Omron CX-Programmer project NewProject (CX-Programmer 9.03)

# PLC CLP: CJ1M CPU11
I/O table (CPU CJ1M-CPU11): rack 0 slot 0 CJ1W-ETN21(ETN11Mode); rack 0 slot 1 CJ1W-ID211; rack 0 slot 2 CJ1W-OD211; rack 0 slot 3 CJ1W-ID211; rack 0 slot 4 CJ1W-OD211; rack 0 slot 5 CJ1W-ID211; rack 0 slot 6 CJ1W-OD232

## Global symbols (name address type ; comment)
AS_RS_Ativado 5.02 BOOL
AS_RS_Eixo_X_Ctrg 5.04 BOOL
AS_RS_Eixo_X_D0 5.05 BOOL
AS_RS_Eixo_X_D1 5.06 BOOL
AS_RS_Eixo_X_D2 5.07 BOOL
AS_RS_Eixo_X_D3 5.08 BOOL
AS_RS_Eixo_X_To_Home 5.03 BOOL
AS_RS_Eixo_Y_Ctrg 5.10 BOOL
AS_RS_Eixo_Y_D0 5.11 BOOL
AS_RS_Eixo_Y_D1 5.12 BOOL
AS_RS_Eixo_Y_D2 5.13 BOOL
AS_RS_Eixo_Y_D3 5.14 BOOL
AS_RS_Eixo_Y_To_Home 5.09 BOOL
AS_RS_Eixo_Z_Ctrg 6.00 BOOL
AS_RS_Eixo_Z_D0 6.01 BOOL
AS_RS_Eixo_Z_D1 6.02 BOOL
AS_RS_Eixo_Z_D2 6.03 BOOL
AS_RS_Eixo_Z_D3 6.04 BOOL
AS_RS_Eixo_Z_To_Home 5.15 BOOL
AS_RS_Home_X_Completo 4.05 BOOL
AS_RS_Home_Y_Completo 4.07 BOOL
AS_RS_Home_Z_Completo 4.09 BOOL
AS_RS_Pos_X_Completa 4.04 BOOL
AS_RS_Pos_Y_Completa 4.06 BOOL
AS_RS_Pos_Z_Completa 4.08 BOOL
AUX_CTRG W10.02 BOOL
AUX_X_OK W10.05 BOOL
AUX_X_OK_DESCIDA W16.00 BOOL
AUX_Y_OK W10.07 BOOL
AUX_Z_OK W10.06 BOOL
AUX_Z_OK_DESCIDA W16.01 BOOL
T0005 BOOL  ; 3
CONF_Z W11.05 BOOL
Confirmacao W4.00 BOOL
Eletroval1 1.06 BOOL
Eletroval2 1.07 BOOL
Eletroval3 1.08 BOOL
Eletroval4 1.09 BOOL
Elevar_Z W15.00 BOOL
Esteira1 1.00 BOOL
Esteira2 1.01 BOOL
Esteira3 1.02 BOOL
Esteira4 1.03 BOOL
Etapa BOOL
Etapa0 W0.00 BOOL
Etapa1 W0.01 BOOL
Etapa10 W1.02 BOOL
Etapa11 W1.03 BOOL
Etapa2 W0.02 BOOL
Etapa3 W0.03 BOOL
Etapa4 W0.04 BOOL
Etapa5 W0.05 BOOL
Etapa6 W0.06 BOOL
Etapa7 W0.07 BOOL
Etapa8 W1.00 BOOL
Etapa9 W1.01 BOOL
Home_X_Completo 4.05 BOOL
Home_Y_Completo 4.07 BOOL
Home_Z_Completo 4.09 BOOL
Pos_X_Completa 4.04 BOOL
Pos_Y_Completa 4.06 BOOL
Pos_Z_Completa 4.08 BOOL
Sensor1 0.00 BOOL
Sensor2 0.01 BOOL
Sensor3 0.02 BOOL
Sensor4 0.03 BOOL
X_CTRG 5.04 BOOL
X_D0 5.05 BOOL
X_D1 5.06 BOOL
X_D2 5.07 BOOL
X_D3 5.08 BOOL
X_To_Home 5.03 BOOL
Y_CTRG 5.10 BOOL
Y_D0 5.11 BOOL
Y_D1 5.12 BOOL
Y_D2 5.13 BOOL
Y_D3 5.14 BOOL
Y_To_Home 5.09 BOOL
Z_CTRG 6.00 BOOL
Z_D0 6.01 BOOL
Z_D1 6.02 BOOL
Z_D2 6.03 BOOL
Z_D3 6.04 BOOL
Z_To_Home 5.15 BOOL

## Program NewProgram1 (cyclic task 0)
Local symbols
AS_RS_Ativado 5.02 BOOL
AUX_CTRG W10.02 BOOL
AUX_ESTEIRA_OK W65.00 BOOL
AUX_ROBO_OK W50.00 BOOL
AUX_VISAO_OK W50.01 BOOL
AUX_X_OK W10.05 BOOL
AUX_Y_OK W10.07 BOOL
AUX_Z_OK W10.06 BOOL
Confirmacao W4.00 BOOL
E0_ESTEIRA W60.00 BOOL
E1_ESTEIRA W60.01 BOOL
E2_ESTEIRA W60.02 BOOL
E3_ESTEIRA W60.03 BOOL
E4_ESTEIRA W60.04 BOOL
E5_ESTEIRA W60.05 BOOL
E6_ESTEIRA W60.06 BOOL
E7_ESTEIRA W60.07 BOOL
Eletroval1 1.06 BOOL
Eletroval2 1.07 BOOL
Eletroval3 1.08 BOOL
Eletroval4 1.09 BOOL
Elevar_Z W15.00 BOOL
Esteira1 1.00 BOOL
Esteira2 1.01 BOOL
Esteira3 1.02 BOOL
Esteira4 1.03 BOOL
Etapa BOOL
Etapa0 W0.00 BOOL
Etapa1 W0.01 BOOL
Etapa10 W1.02 BOOL
Etapa11 W1.03 BOOL
Etapa12 W1.04 BOOL
Etapa13 W1.05 BOOL
Etapa14 W1.06 BOOL
Etapa15 W1.07 BOOL
Etapa16 W2.00 BOOL
Etapa17 W2.01 BOOL
Etapa18 W2.02 BOOL
Etapa19 W2.03 BOOL
Etapa2 W0.02 BOOL
Etapa20 W2.04 BOOL
Etapa21 W2.05 BOOL
Etapa22 W2.06 BOOL
Etapa23 W2.07 BOOL
Etapa24 W3.01 BOOL
Etapa25 W3.02 BOOL
Etapa26 W3.03 BOOL
Etapa27 W3.04 BOOL
Etapa28 W3.05 BOOL
Etapa29 W3.06 BOOL
Etapa3 W0.03 BOOL
Etapa30 W3.07 BOOL
Etapa31 W4.01 BOOL
Etapa32 W4.02 BOOL
Etapa33 W4.03 BOOL
Etapa34 W4.04 BOOL
Etapa35 W4.05 BOOL
Etapa36 W4.06 BOOL
Etapa4 W0.04 BOOL
Etapa5 W0.05 BOOL
Etapa6 W0.06 BOOL
Etapa7 W0.07 BOOL
Etapa8 W1.00 BOOL
Etapa9 W1.01 BOOL
FLAG_ROBO W50.02 BOOL
Home_X_Completo 4.05 BOOL
Home_Y_Completo 4.07 BOOL
Home_Z_Completo 4.09 BOOL
INICIA_ESTEIRA BOOL
INICIA_ESTEIRAS W50.05 BOOL
MAO_PEGAR_ARMAZEM 6.08 BOOL
MAO_PEGAR_ESTEIRA 6.09 BOOL
PEGAR_MAO_ESTEIRA BOOL
Pos_X_Completa 4.04 BOOL
Pos_Y_Completa 4.06 BOOL
Pos_Z_Completa 4.08 BOOL
Sensor1 0.00 BOOL
Sensor2 0.01 BOOL
Sensor3 0.02 BOOL
Sensor4 0.03 BOOL
WORD_X W35 WORD
WORD_Z W40 WORD
XD0 BOOL
X_CTRG 5.04 BOOL
X_D0 5.05 BOOL
X_D1 5.06 BOOL
X_D2 5.07 BOOL
X_D3 5.08 BOOL
X_To_Home 5.03 BOOL
Y_CTRG 5.10 BOOL
Y_D0 5.11 BOOL
Y_D1 5.12 BOOL
Y_D2 5.13 BOOL
Y_D3 5.14 BOOL
Y_To_Home 5.09 BOOL
Z_CTRG 6.00 BOOL
Z_D0 6.01 BOOL
Z_D1 6.02 BOOL
Z_D2 6.03 BOOL
Z_D3 6.04 BOOL
Z_To_Home 5.15 BOOL

### Section Armazem

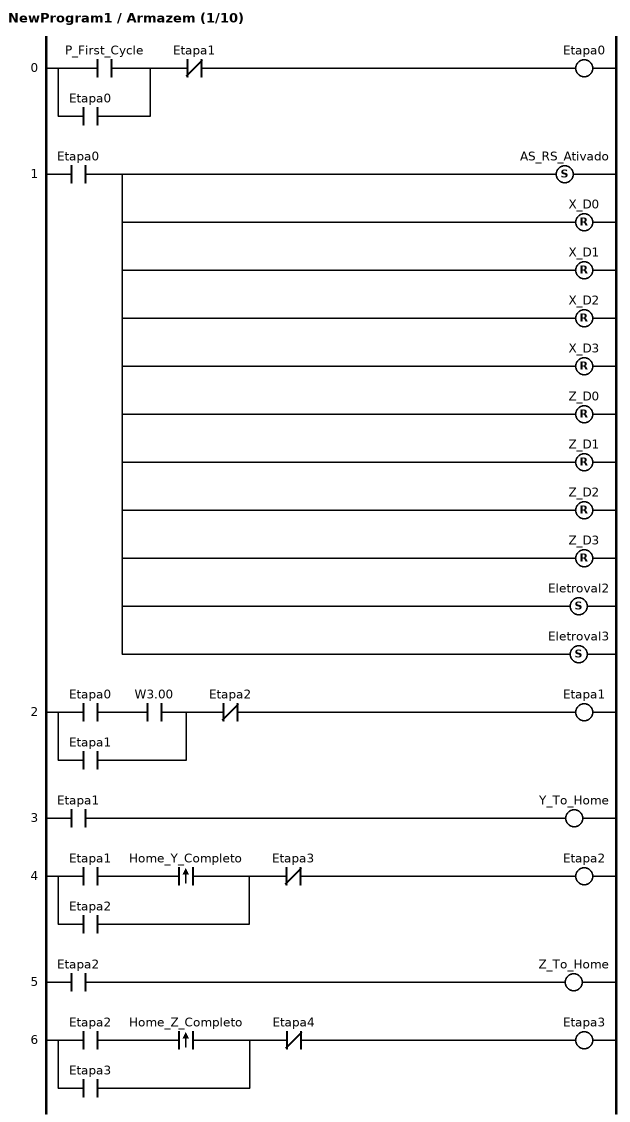
; rung 0
LD P_First_Cycle
OR Etapa0
ANDNOT Etapa1
OUT Etapa0
; rung 1
LD Etapa0
SET AS_RS_Ativado
RSET X_D0
RSET X_D1
RSET X_D2
RSET X_D3
RSET Z_D0
RSET Z_D1
RSET Z_D2
RSET Z_D3
SET Eletroval2
SET Eletroval3
; rung 2
LD Etapa0
AND W3.00
OR Etapa1
ANDNOT Etapa2
OUT Etapa1
; rung 3
LD Etapa1
OUT Y_To_Home
; rung 4
LD Etapa1
@AND Home_Y_Completo
OR Etapa2
ANDNOT Etapa3
OUT Etapa2
; rung 5
LD Etapa2
OUT Z_To_Home
; rung 6
LD Etapa2
@AND Home_Z_Completo
OR Etapa3
ANDNOT Etapa4
OUT Etapa3

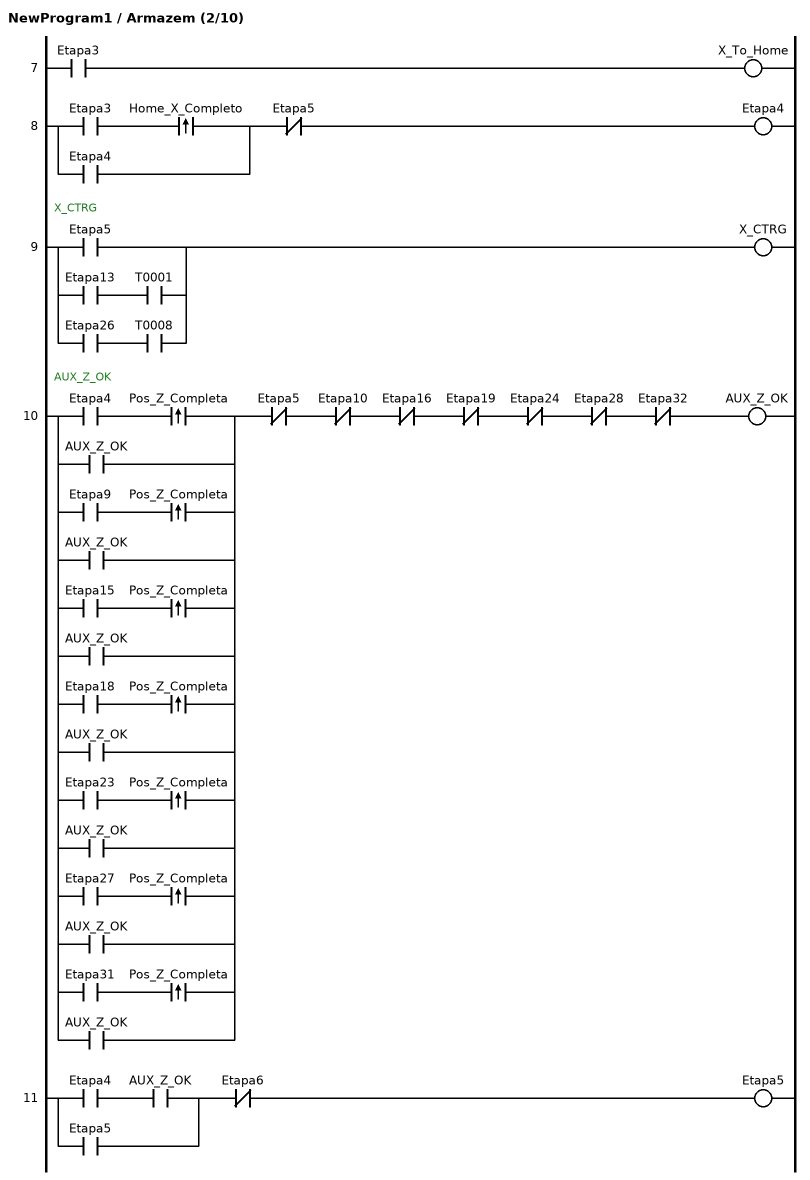
; rung 7
LD Etapa3
OUT X_To_Home
; rung 8
LD Etapa3
@AND Home_X_Completo
OR Etapa4
ANDNOT Etapa5
OUT Etapa4
; rung 9: X_CTRG
LD Etapa5
LD Etapa13
AND T0001
ORLD
LD Etapa26
AND T0008
ORLD
OUT X_CTRG
; rung 10: AUX_Z_OK
LD Etapa4
@AND Pos_Z_Completa
OR AUX_Z_OK
LD Etapa9
@AND Pos_Z_Completa
ORLD
OR AUX_Z_OK
LD Etapa15
@AND Pos_Z_Completa
ORLD
OR AUX_Z_OK
LD Etapa18
@AND Pos_Z_Completa
ORLD
OR AUX_Z_OK
LD Etapa23
@AND Pos_Z_Completa
ORLD
OR AUX_Z_OK
LD Etapa27
@AND Pos_Z_Completa
ORLD
OR AUX_Z_OK
LD Etapa31
@AND Pos_Z_Completa
ORLD
OR AUX_Z_OK
ANDNOT Etapa5
ANDNOT Etapa10
ANDNOT Etapa16
ANDNOT Etapa19
ANDNOT Etapa24
ANDNOT Etapa28
ANDNOT Etapa32
OUT AUX_Z_OK
; rung 11
LD Etapa4
AND AUX_Z_OK
OR Etapa5
ANDNOT Etapa6
OUT Etapa5

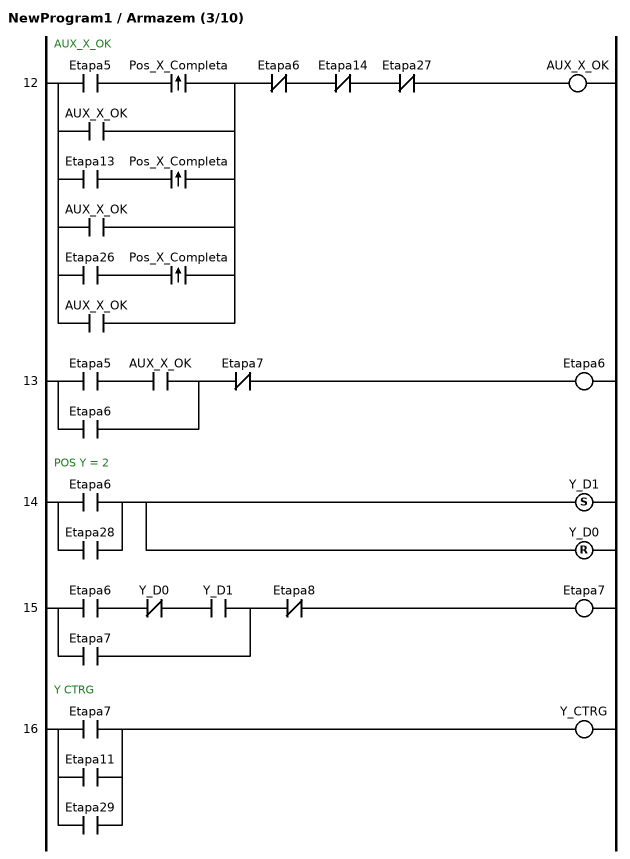
; rung 12: AUX_X_OK
LD Etapa5
@AND Pos_X_Completa
OR AUX_X_OK
LD Etapa13
@AND Pos_X_Completa
ORLD
OR AUX_X_OK
LD Etapa26
@AND Pos_X_Completa
ORLD
OR AUX_X_OK
ANDNOT Etapa6
ANDNOT Etapa14
ANDNOT Etapa27
OUT AUX_X_OK
; rung 13
LD Etapa5
AND AUX_X_OK
OR Etapa6
ANDNOT Etapa7
OUT Etapa6
; rung 14: POS Y = 2
LD Etapa6
OR Etapa28
SET Y_D1
RSET Y_D0
; rung 15
LD Etapa6
ANDNOT Y_D0
AND Y_D1
OR Etapa7
ANDNOT Etapa8
OUT Etapa7
; rung 16: Y CTRG
LD Etapa7
OR Etapa11
OR Etapa29
OUT Y_CTRG

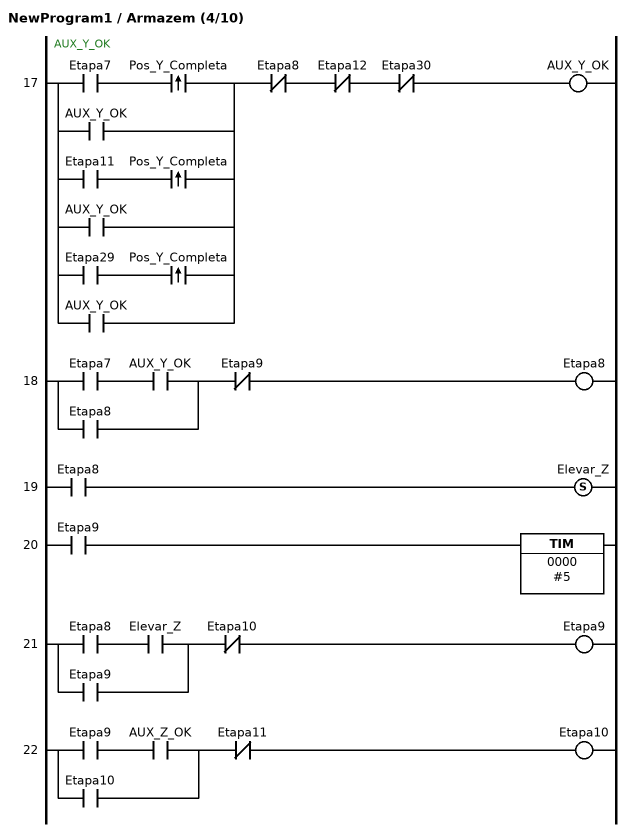
; rung 17: AUX_Y_OK
LD Etapa7
@AND Pos_Y_Completa
OR AUX_Y_OK
LD Etapa11
@AND Pos_Y_Completa
ORLD
OR AUX_Y_OK
LD Etapa29
@AND Pos_Y_Completa
ORLD
OR AUX_Y_OK
ANDNOT Etapa8
ANDNOT Etapa12
ANDNOT Etapa30
OUT AUX_Y_OK
; rung 18
LD Etapa7
AND AUX_Y_OK
OR Etapa8
ANDNOT Etapa9
OUT Etapa8
; rung 19
LD Etapa8
SET Elevar_Z
; rung 20
LD Etapa9
TIM 0000 #5
; rung 21
LD Etapa8
AND Elevar_Z
OR Etapa9
ANDNOT Etapa10
OUT Etapa9
; rung 22
LD Etapa9
AND AUX_Z_OK
OR Etapa10
ANDNOT Etapa11
OUT Etapa10

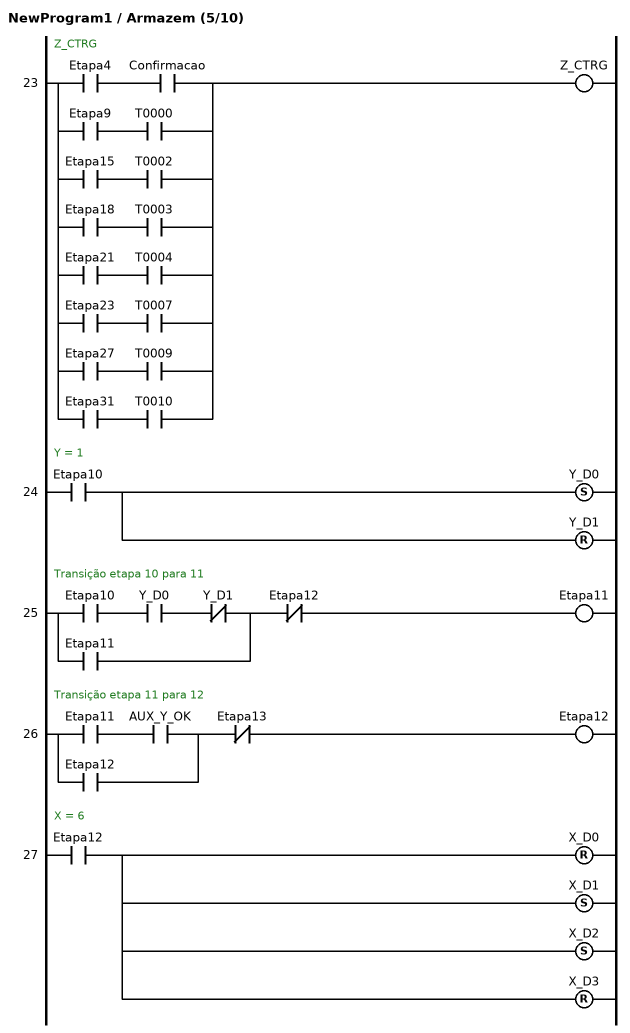
; rung 23: Z_CTRG
LD Etapa4
AND Confirmacao
LD Etapa9
AND T0000
ORLD
LD Etapa15
AND T0002
ORLD
LD Etapa18
AND T0003
ORLD
LD Etapa21
AND T0004
ORLD
LD Etapa23
AND T0007
ORLD
LD Etapa27
AND T0009
ORLD
LD Etapa31
AND T0010
ORLD
OUT Z_CTRG
; rung 24: Y = 1
LD Etapa10
SET Y_D0
RSET Y_D1
; rung 25: Transição etapa 10 para 11
LD Etapa10
AND Y_D0
ANDNOT Y_D1
OR Etapa11
ANDNOT Etapa12
OUT Etapa11
; rung 26: Transição etapa 11 para 12
LD Etapa11
AND AUX_Y_OK
OR Etapa12
ANDNOT Etapa13
OUT Etapa12
; rung 27: X = 6
LD Etapa12
RSET X_D0
SET X_D1
SET X_D2
RSET X_D3

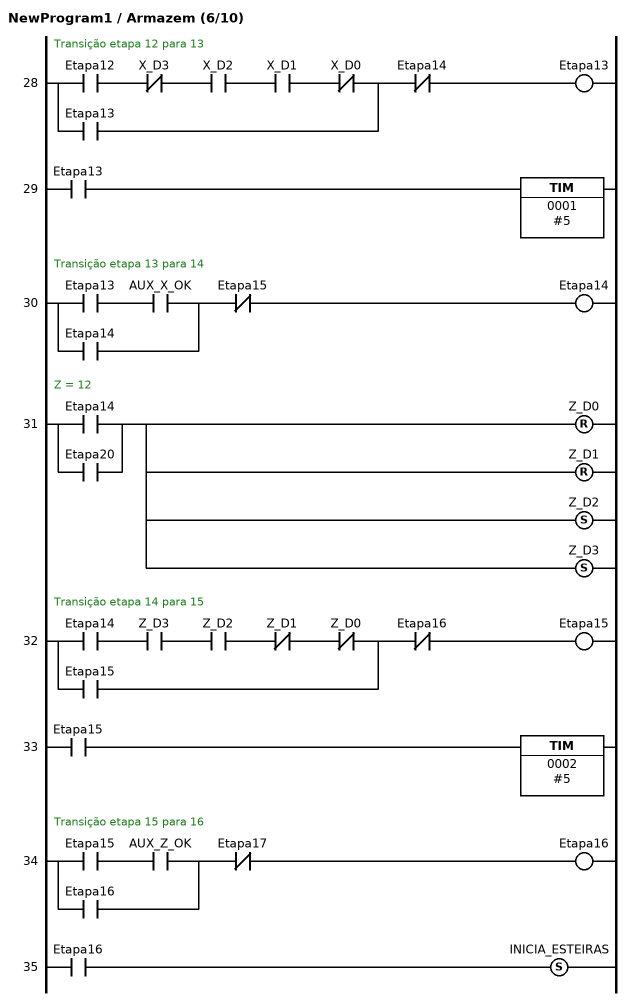
; rung 28: Transição etapa 12 para 13
LD Etapa12
ANDNOT X_D3
AND X_D2
AND X_D1
ANDNOT X_D0
OR Etapa13
ANDNOT Etapa14
OUT Etapa13
; rung 29
LD Etapa13
TIM 0001 #5
; rung 30: Transição etapa 13 para 14
LD Etapa13
AND AUX_X_OK
OR Etapa14
ANDNOT Etapa15
OUT Etapa14
; rung 31: Z = 12
LD Etapa14
OR Etapa20
RSET Z_D0
RSET Z_D1
SET Z_D2
SET Z_D3
; rung 32: Transição etapa 14 para 15
LD Etapa14
AND Z_D3
AND Z_D2
ANDNOT Z_D1
ANDNOT Z_D0
OR Etapa15
ANDNOT Etapa16
OUT Etapa15
; rung 33
LD Etapa15
TIM 0002 #5
; rung 34: Transição etapa 15 para 16
LD Etapa15
AND AUX_Z_OK
OR Etapa16
ANDNOT Etapa17
OUT Etapa16
; rung 35
LD Etapa16
SET INICIA_ESTEIRAS

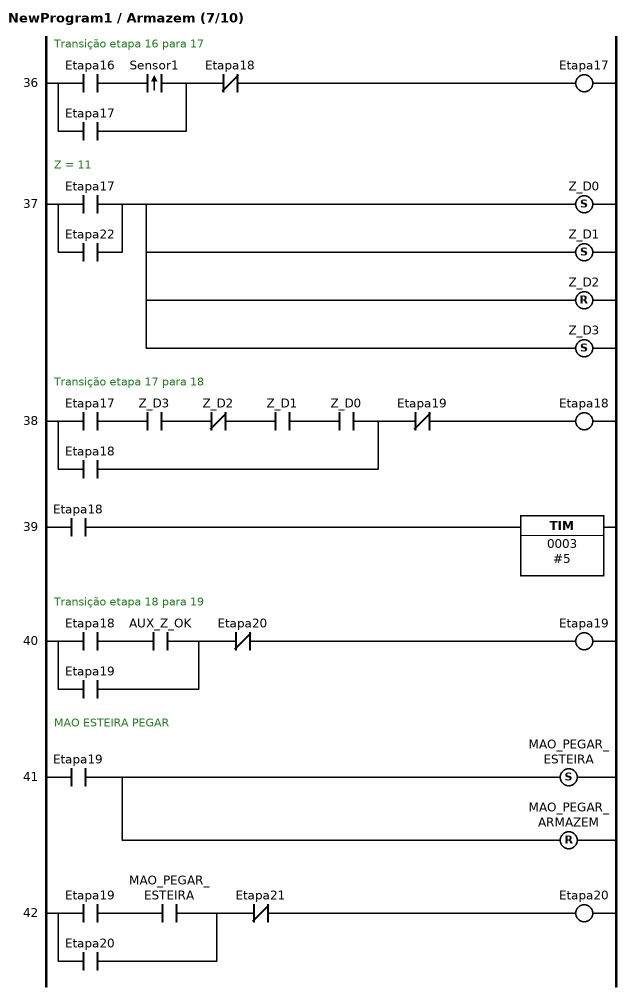
; rung 36: Transição etapa 16 para 17
LD Etapa16
@AND Sensor1
OR Etapa17
ANDNOT Etapa18
OUT Etapa17
; rung 37: Z = 11
LD Etapa17
OR Etapa22
SET Z_D0
SET Z_D1
RSET Z_D2
SET Z_D3
; rung 38: Transição etapa 17 para 18
LD Etapa17
AND Z_D3
ANDNOT Z_D2
AND Z_D1
AND Z_D0
OR Etapa18
ANDNOT Etapa19
OUT Etapa18
; rung 39
LD Etapa18
TIM 0003 #5
; rung 40: Transição etapa 18 para 19
LD Etapa18
AND AUX_Z_OK
OR Etapa19
ANDNOT Etapa20
OUT Etapa19
; rung 41: MAO ESTEIRA PEGAR
LD Etapa19
SET MAO_PEGAR_ESTEIRA
RSET MAO_PEGAR_ARMAZEM
; rung 42
LD Etapa19
AND MAO_PEGAR_ESTEIRA
OR Etapa20
ANDNOT Etapa21
OUT Etapa20
; rung 43: MAO ARMAZEM PEGAR

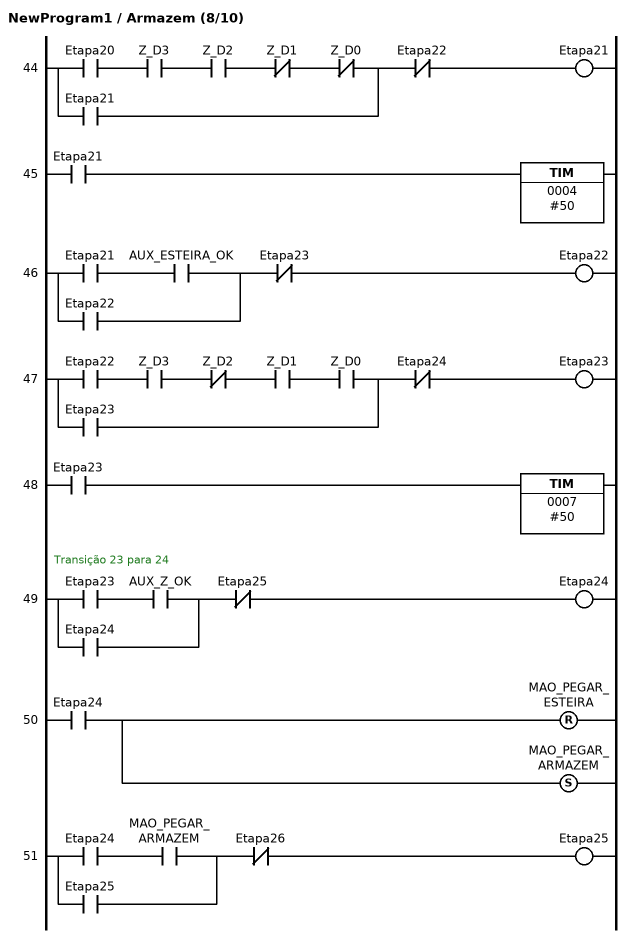
; rung 44
LD Etapa20
AND Z_D3
AND Z_D2
ANDNOT Z_D1
ANDNOT Z_D0
OR Etapa21
ANDNOT Etapa22
OUT Etapa21
; rung 45
LD Etapa21
TIM 0004 #50
; rung 46
LD Etapa21
AND AUX_ESTEIRA_OK
OR Etapa22
ANDNOT Etapa23
OUT Etapa22
; rung 47
LD Etapa22
AND Z_D3
ANDNOT Z_D2
AND Z_D1
AND Z_D0
OR Etapa23
ANDNOT Etapa24
OUT Etapa23
; rung 48
LD Etapa23
TIM 0007 #50
; rung 49: Transição 23 para 24
LD Etapa23
AND AUX_Z_OK
OR Etapa24
ANDNOT Etapa25
OUT Etapa24
; rung 50
LD Etapa24
RSET MAO_PEGAR_ESTEIRA
SET MAO_PEGAR_ARMAZEM
; rung 51
LD Etapa24
AND MAO_PEGAR_ARMAZEM
OR Etapa25
ANDNOT Etapa26
OUT Etapa25

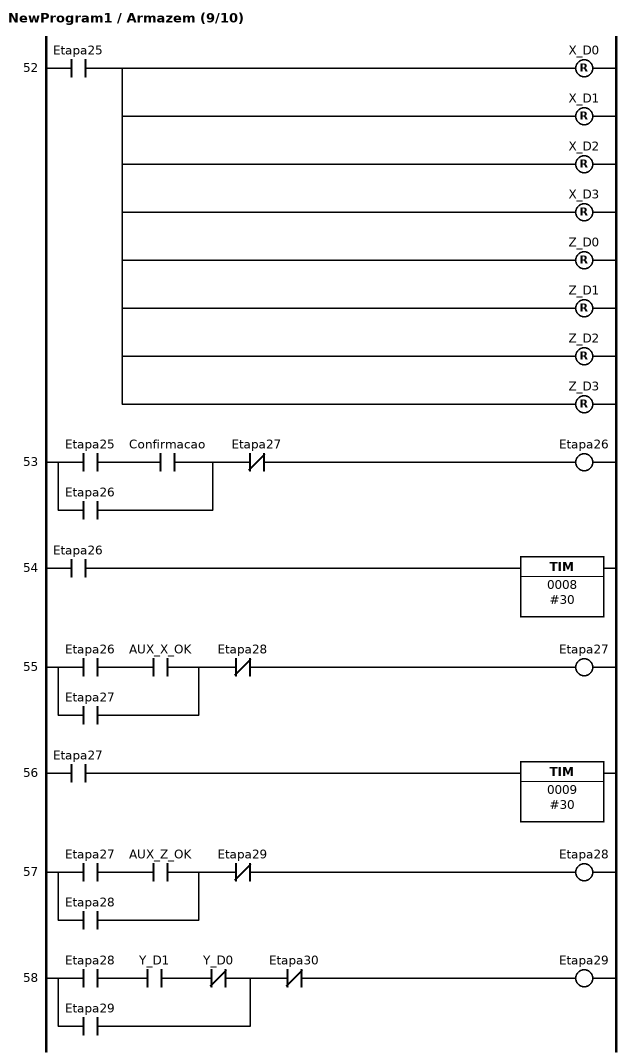
; rung 52
LD Etapa25
RSET X_D0
RSET X_D1
RSET X_D2
RSET X_D3
RSET Z_D0
RSET Z_D1
RSET Z_D2
RSET Z_D3
; rung 53
LD Etapa25
AND Confirmacao
OR Etapa26
ANDNOT Etapa27
OUT Etapa26
; rung 54
LD Etapa26
TIM 0008 #30
; rung 55
LD Etapa26
AND AUX_X_OK
OR Etapa27
ANDNOT Etapa28
OUT Etapa27
; rung 56
LD Etapa27
TIM 0009 #30
; rung 57
LD Etapa27
AND AUX_Z_OK
OR Etapa28
ANDNOT Etapa29
OUT Etapa28
; rung 58
LD Etapa28
AND Y_D1
ANDNOT Y_D0
OR Etapa29
ANDNOT Etapa30
OUT Etapa29

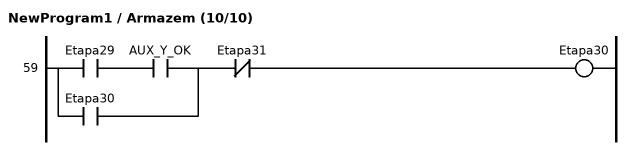
; rung 59
LD Etapa29
AND AUX_Y_OK
OR Etapa30
ANDNOT Etapa31
OUT Etapa30

### Section Robo

### Section Visao

### Section Esteiras

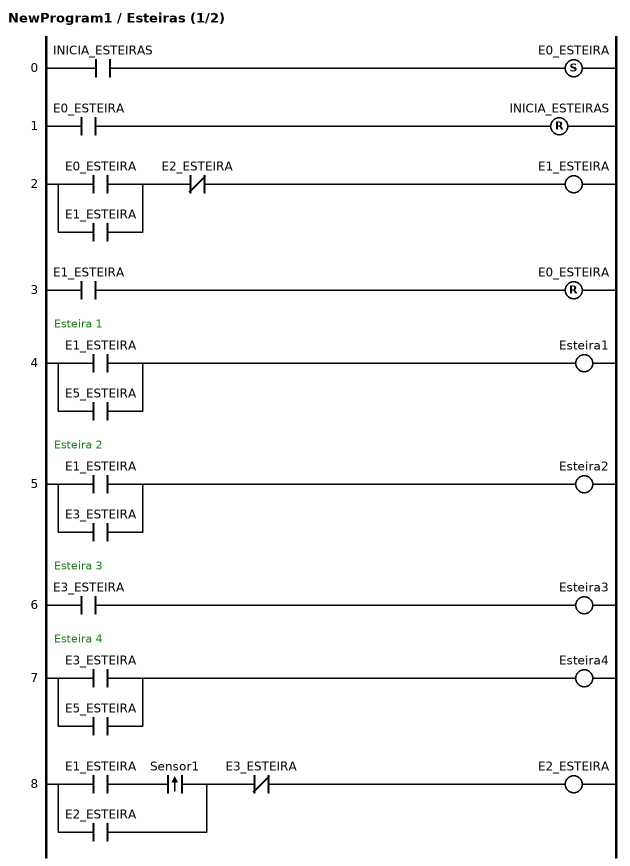
; rung 0
LD INICIA_ESTEIRAS
SET E0_ESTEIRA
; rung 1
LD E0_ESTEIRA
RSET INICIA_ESTEIRAS
; rung 2
LD E0_ESTEIRA
OR E1_ESTEIRA
ANDNOT E2_ESTEIRA
OUT E1_ESTEIRA
; rung 3
LD E1_ESTEIRA
RSET E0_ESTEIRA
; rung 4: Esteira 1
LD E1_ESTEIRA
OR E5_ESTEIRA
OUT Esteira1
; rung 5: Esteira 2
LD E1_ESTEIRA
OR E3_ESTEIRA
OUT Esteira2
; rung 6: Esteira 3
LD E3_ESTEIRA
OUT Esteira3
; rung 7: Esteira 4
LD E3_ESTEIRA
OR E5_ESTEIRA
OUT Esteira4
; rung 8
LD E1_ESTEIRA
@AND Sensor1
OR E2_ESTEIRA
ANDNOT E3_ESTEIRA
OUT E2_ESTEIRA

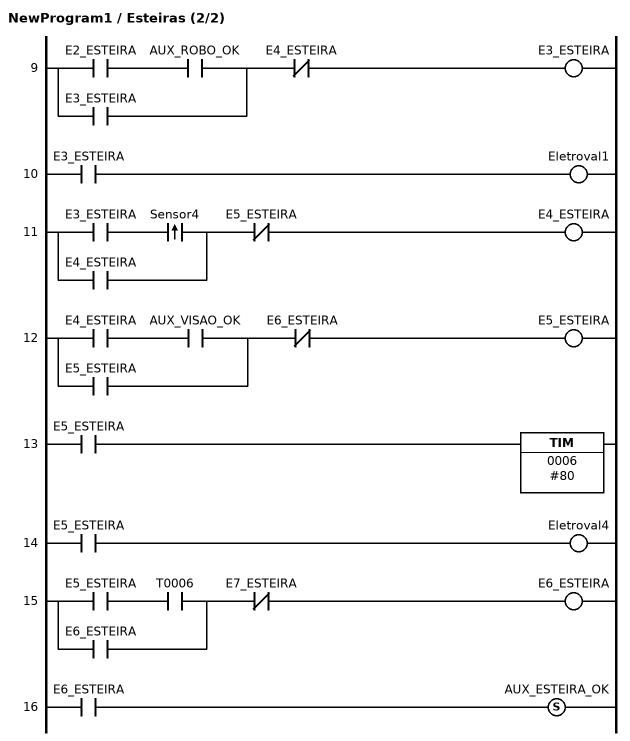
; rung 9
LD E2_ESTEIRA
AND AUX_ROBO_OK
OR E3_ESTEIRA
ANDNOT E4_ESTEIRA
OUT E3_ESTEIRA
; rung 10
LD E3_ESTEIRA
OUT Eletroval1
; rung 11
LD E3_ESTEIRA
@AND Sensor4
OR E4_ESTEIRA
ANDNOT E5_ESTEIRA
OUT E4_ESTEIRA
; rung 12
LD E4_ESTEIRA
AND AUX_VISAO_OK
OR E5_ESTEIRA
ANDNOT E6_ESTEIRA
OUT E5_ESTEIRA
; rung 13
LD E5_ESTEIRA
TIM 0006 #80
; rung 14
LD E5_ESTEIRA
OUT Eletroval4
; rung 15
LD E5_ESTEIRA
AND T0006
OR E6_ESTEIRA
ANDNOT E7_ESTEIRA
OUT E6_ESTEIRA
; rung 16
LD E6_ESTEIRA
SET AUX_ESTEIRA_OK

### Section END
; rung 0
END(001)